FUNCTION_BLOCK MotorPPScheduler
VAR
	_skd_state: motor_pp_states_t:=motor_pp_states_t.END;
	_profile_velocity: UDINT:= 10000;
	_profile_acceleration: UDINT:= 300000;
	
	_change_immediately: BOOL;
	_reference_coordinate: BOOL;
	_push_operation: BOOL;
	
	_target_position: DINT;
	_motor_interface_adr: POINTER TO MotorInterface;
	
	_statusword: UINT;
	_controlword_adr : POINTER TO UINT;
	_last_send_time: ULINT;
	_MSG_SENT:BOOL:=FALSE;
END_VAR

IF _motor_interface_adr^.driver_mode=driver_modes_t.PP AND _motor_interface_adr^.driver_enable AND _motor_interface_adr^.driver_state<>driver_states_t.Fault AND _motor_interface_adr^.driver_state<>driver_states_t.FaultReactionActive THEN
	_statusword := _motor_interface_adr^.statusword;
	_motor_interface_adr^.set_PP_parameters(profile_velocity:=_profile_velocity, profile_acceleration:=_profile_acceleration);
	_controlword_adr^.5:=_change_immediately;
	_controlword_adr^.6:=_reference_coordinate;
	_controlword_adr^.13:=_push_operation;
	
	CASE _skd_state OF
		motor_pp_states_t.START: 
			_skd_state:=motor_pp_states_t.SENDINGCMD;
			_controlword_adr^.4:=0;
			_MSG_SENT:=FALSE;
		motor_pp_states_t.SENDINGCMD:
			_controlword_adr^.4:=1;
			IF NOT _MSG_SENT THEN
				_last_send_time:=SYSTIME_MS();
			END_IF
			_MSG_SENT:=TRUE;
			IF _statusword.12 THEN
				_skd_state := motor_pp_states_t.INPROGRESS;
			ELSIF (SYSTIME_MS()-_last_send_time)>500 THEN
				_MSG_SENT:=FALSE;
				_controlword_adr^.4:=0;
			END_IF
		motor_pp_states_t.INPROGRESS:
			_controlword_adr^.4:=1;
			// 10 is end to target, while 15 is reaches to torque limit (limited by mechanical structure)
			IF _statusword.10 OR _statusword.15 THEN
				_skd_state := motor_pp_states_t.END;
			END_IF
		motor_pp_states_t.END:
			_controlword_adr^.4:=0;
	END_CASE
	_motor_interface_adr^.target_position:=_target_position;
END_IF

METHOD activate : BOOL
VAR_INPUT
END_VAR
_motor_interface_adr^.driver_mode:=driver_modes_t.PP;
END_METHOD

METHOD FB_init : BOOL
VAR_INPUT
	bInitRetains : BOOL; // if TRUE, the retain variables are initialized (warm start / cold start)
	bInCopyCode : BOOL;  // if TRUE, the instance afterwards gets moved into the copy code (online change)
	motor_interface_adr : POINTER TO MotorInterface;
END_VAR
_motor_interface_adr := motor_interface_adr;
_controlword_adr := _motor_interface_adr^.controlword_adr;
END_METHOD

{attribute 'TcRpcEnable'}
METHOD get_state : motor_pp_states_t
VAR_INPUT
END_VAR
get_state:=_skd_state;
END_METHOD

{attribute 'TcRpcEnable'}
METHOD start_operation : BOOL
VAR_INPUT
	target_position: LINT;
	change_immediately: BOOL;
	reference_coordinate: BOOL;
	push_operation: BOOL;
END_VAR
_change_immediately:=change_immediately;
_reference_coordinate:=reference_coordinate;
_push_operation:=push_operation;
IF(reference_coordinate) THEN
	_target_position := TO_DINT(target_position);
ELSE
	_target_position := TO_DINT(target_position - _motor_interface_adr^.feedback_position + _motor_interface_adr^.raw_position);
END_IF
_skd_state:=motor_pp_states_t.START;
END_METHOD

METHOD update_pp_parameter : BOOL
VAR_INPUT
	profile_velocity:UDINT;
	profile_acceleration:UDINT;
END_VAR
_profile_velocity:=profile_velocity;
_profile_acceleration:=profile_acceleration;
END_METHOD

END_FUNCTION_BLOCK

(* stored: Version 1.1.0.1, ProductVersion 3.1.4024.12
   POU MotorPPScheduler: Id {33dfd4c6-4195-41e6-9061-13970559ee38}, SpecialFunc None
   Method activate: Id {ccf61a8c-f1c3-4a4b-9059-6aed63841325}
   Method FB_init: Id {24ceeb3a-84c3-4cde-8b7e-80d2cf7a268f}
   Method get_state: Id {66669643-288f-4ab7-b584-70451d57dbaf}
   Method start_operation: Id {b514f046-fed4-432d-bdf7-dc77a1ac8372}
   Method update_pp_parameter: Id {f4219e36-5ad5-430a-9db8-b0d5c64f626a} *)
